// TIA Portal V18 export
// export: Created 2026-06-22T00:00:00Z, ExportSetting WithDefaults, DisplayName Totally Integrated Automation Portal, DisplayVersion V18
TagTable "Default tag table"
  CV3201_Nuoc_Bon1_M : Real  (PLC tag CV3201_Nuoc_Bon1_M, HMI_Connection_1, 1 s)   // Cảm biến/Van tuyến tính CV 32.01
  CV3206_Hoi_Bon2_M : Real  (PLC tag CV3206_Hoi_Bon2_M, HMI_Connection_1, 1 s)   // Cảm biến/Van tuyến tính CV 32.06
  CV3211_Nuoc_Bon3_M : Real  (PLC tag CV3211_Nuoc_Bon3_M, HMI_Connection_1, 1 s)   // Cảm biến/Van tuyến tính CV 32.11
  CV3216_Hoi_Bon4_M : Real  (PLC tag CV3216_Hoi_Bon4_M, HMI_Connection_1, 1 s)   // Cảm biến/Van tuyến tính CV 32.16
  CV3304_Nuoc_Lam_Mat_M : Real  (PLC tag CV3304_Nuoc_Lam_Mat_M, HMI_Connection_1, 1 s)   // Cảm biến/Van tuyến tính CV 33.04
  CV_Filler_Cap_Dich_M : Real  (PLC tag CV_Filler_Cap_Dich_M, HMI_Connection_1, 1 s)   // Cảm biến/Van tuyến tính CV Filler
  FQ3200_Bon1_Eff : Real  (PLC tag FQ3200_Bon1_Eff, HMI_Connection_1, 1 s)   // Cảm biến/Van tuyến tính FT 32.00
  FQ3205_Bon2_Eff : Real  (PLC tag FQ3205_Bon2_Eff, HMI_Connection_1, 1 s)   // Cảm biến/Van tuyến tính FT 32.05
  FQ3210_Bon3_Eff : Real  (PLC tag FQ3210_Bon3_Eff, HMI_Connection_1, 1 s)   // Cảm biến/Van tuyến tính FT 32.10
  FQ3215_Bon4_Eff : Real  (PLC tag FQ3215_Bon4_Eff, HMI_Connection_1, 1 s)   // Cảm biến/Van tuyến tính FT 32.15
  FT3309_Xa_Thanh_Pham_Eff : Real  (PLC tag FT3309_Xa_Thanh_Pham_Eff, HMI_Connection_1, 1 s)   // Cảm biến/Van tuyến tính FT 33.09
  HMI_Anim_Bon1_Frame : Int  (PLC tag HMI_Anim_Bon1_Frame, HMI_Connection_1, 1 s)   // Trạng thái hoạt hình HMI HMI_Anim_Bon1_Frame
  HMI_Anim_Bon1_MucDich : Int  (PLC tag HMI_Anim_Bon1_MucDich, HMI_Connection_1, 1 s)   // Trạng thái hoạt hình HMI HMI_Anim_Bon1_MucDich
  HMI_Anim_Bon2_Frame : Int  (PLC tag HMI_Anim_Bon2_Frame, HMI_Connection_1, 1 s)   // Trạng thái hoạt hình HMI HMI_Anim_Bon2_Frame
  HMI_Anim_Bon2_MucDich : Int  (PLC tag HMI_Anim_Bon2_MucDich, HMI_Connection_1, 1 s)   // Trạng thái hoạt hình HMI HMI_Anim_Bon2_MucDich
  HMI_Anim_Bon3_Frame : Int  (PLC tag HMI_Anim_Bon3_Frame, HMI_Connection_1, 1 s)   // Trạng thái hoạt hình HMI HMI_Anim_Bon3_Frame
  HMI_Anim_Bon3_MucDich : Int  (PLC tag HMI_Anim_Bon3_MucDich, HMI_Connection_1, 1 s)   // Trạng thái hoạt hình HMI HMI_Anim_Bon3_MucDich
  HMI_Anim_Bon4_Frame : Int  (PLC tag HMI_Anim_Bon4_Frame, HMI_Connection_1, 1 s)   // Trạng thái hoạt hình HMI HMI_Anim_Bon4_Frame
  HMI_Anim_Bon4_MucDich : Int  (PLC tag HMI_Anim_Bon4_MucDich, HMI_Connection_1, 1 s)   // Trạng thái hoạt hình HMI HMI_Anim_Bon4_MucDich
  HMI_Anim_BonChua1_MucDich : Int  (PLC tag HMI_Anim_BonChua1_MucDich, HMI_Connection_1, 1 s)   // Trạng thái hoạt hình HMI HMI_Anim_BonChua1_MucDich
  HMI_Anim_BonChua2_MucDich : Int  (PLC tag HMI_Anim_BonChua2_MucDich, HMI_Connection_1, 1 s)   // Trạng thái hoạt hình HMI HMI_Anim_BonChua2_MucDich
  LT3203_Bon1_Eff : Real  (PLC tag LT3203_Bon1_Eff, HMI_Connection_1, 1 s)   // Cảm biến/Van tuyến tính LT 32.03
  LT3209_Bon2_Eff : Real  (PLC tag LT3209_Bon2_Eff, HMI_Connection_1, 1 s)   // Cảm biến/Van tuyến tính LT 32.09
  LT3213_Bon3_Eff : Real  (PLC tag LT3213_Bon3_Eff, HMI_Connection_1, 1 s)   // Cảm biến/Van tuyến tính LT 32.13
  LT3218_Bon4_Eff : Real  (PLC tag LT3218_Bon4_Eff, HMI_Connection_1, 1 s)   // Cảm biến/Van tuyến tính LT 32.18
  LT3302_BonChua1_Eff : Real  (PLC tag LT3302_BonChua1_Eff, HMI_Connection_1, 1 s)   // Cảm biến/Van tuyến tính LT 33.02
  LT3307_BonChua2_Eff : Real  (PLC tag LT3307_BonChua2_Eff, HMI_Connection_1, 1 s)   // Cảm biến/Van tuyến tính LT 33.07
  PI3308_Truoc_Filter_Eff : Real  (PLC tag PI3308_Truoc_Filter_Eff, HMI_Connection_1, 1 s)   // Cảm biến/Van tuyến tính PI 33.08
  Pump3264_Chuyen_Nhanh1_M : Bool  (PLC tag Pump3264_Chuyen_Nhanh1_M, HMI_Connection_1, 1 s)   // Trạng thái hoạt động Pump 32.64
  Pump3265_Chuyen_Nhanh2_M : Bool  (PLC tag Pump3265_Chuyen_Nhanh2_M, HMI_Connection_1, 1 s)   // Trạng thái hoạt động Pump 32.69
  Pump3361_LuanChuyen_BonChua1_M : Bool  (PLC tag Pump3361_LuanChuyen_BonChua1_M, HMI_Connection_1, 1 s)   // Trạng thái hoạt động Pump 33.61
  Pump3362_Xa_BonChua1_M : Bool  (PLC tag Pump3362_Xa_BonChua1_M, HMI_Connection_1, 1 s)   // Trạng thái hoạt động Pump 33.62
  Pump3364_Filter_M : Bool  (PLC tag Pump3364_Filter_M, HMI_Connection_1, 1 s)   // Trạng thái hoạt động Pump 33.64
  Pump3365_Filter_M : Bool  (PLC tag Pump3365_Filter_M, HMI_Connection_1, 1 s)   // Trạng thái hoạt động Pump 33.65
  TT3204_Bon1_Eff : Real  (PLC tag TT3204_Bon1_Eff, HMI_Connection_1, 1 s)   // Cảm biến/Van tuyến tính TT 32.04
  TT3208_Bon2_Eff : Real  (PLC tag TT3208_Bon2_Eff, HMI_Connection_1, 1 s)   // Cảm biến/Van tuyến tính TT 32.08
  TT3214_Bon3_Eff : Real  (PLC tag TT3214_Bon3_Eff, HMI_Connection_1, 1 s)   // Cảm biến/Van tuyến tính TT 32.14
  TT3219_Bon4_Eff : Real  (PLC tag TT3219_Bon4_Eff, HMI_Connection_1, 1 s)   // Cảm biến/Van tuyến tính TT 32.19
  TT3301_BonChua1_Eff : Real  (PLC tag TT3301_BonChua1_Eff, HMI_Connection_1, 1 s)   // Cảm biến/Van tuyến tính TT 33.01
  TT3303_TraoDoiNhiet_Eff : Real  (PLC tag TT3303_TraoDoiNhiet_Eff, HMI_Connection_1, 1 s)   // Cảm biến/Van tuyến tính TT 33.03
  TT3306_BonChua2_Eff : Real  (PLC tag TT3306_BonChua2_Eff, HMI_Connection_1, 1 s)   // Cảm biến/Van tuyến tính TT 33.06
  V3230_Nuoc_Bon1_M : Bool  (PLC tag V3230_Nuoc_Bon1_M, HMI_Connection_1, 1 s)   // Trạng thái hoạt động V32.30
  V3232_Xa_Bon1_M : Bool  (PLC tag V3232_Xa_Bon1_M, HMI_Connection_1, 1 s)   // Trạng thái hoạt động V32.32
  V3233_Xa_Bon1_M : Bool  (PLC tag V3233_Xa_Bon1_M, HMI_Connection_1, 1 s)   // Trạng thái hoạt động V32.33
  V3234_Xa_Bon1_M : Bool  (PLC tag V3234_Xa_Bon1_M, HMI_Connection_1, 1 s)   // Trạng thái hoạt động V32.34
  V3235_Nuoc_Bon2_M : Bool  (PLC tag V3235_Nuoc_Bon2_M, HMI_Connection_1, 1 s)   // Trạng thái hoạt động V32.35
  V3237_Xa_Bon2_M : Bool  (PLC tag V3237_Xa_Bon2_M, HMI_Connection_1, 1 s)   // Trạng thái hoạt động V32.37
  V3238_Xa_Bon2_M : Bool  (PLC tag V3238_Xa_Bon2_M, HMI_Connection_1, 1 s)   // Trạng thái hoạt động V32.38
  V3239_Xa_Bon2_M : Bool  (PLC tag V3239_Xa_Bon2_M, HMI_Connection_1, 1 s)   // Trạng thái hoạt động V32.39
  V3240_Nuoc_Bon3_M : Bool  (PLC tag V3240_Nuoc_Bon3_M, HMI_Connection_1, 1 s)   // Trạng thái hoạt động V32.40
  V3242_Xa_Bon3_M : Bool  (PLC tag V3242_Xa_Bon3_M, HMI_Connection_1, 1 s)   // Trạng thái hoạt động V32.42
  V3243_Xa_Bon3_M : Bool  (PLC tag V3243_Xa_Bon3_M, HMI_Connection_1, 1 s)   // Trạng thái hoạt động V32.43
  V3244_Xa_Bon3_M : Bool  (PLC tag V3244_Xa_Bon3_M, HMI_Connection_1, 1 s)   // Trạng thái hoạt động V32.44
  V3245_Nuoc_Bon4_M : Bool  (PLC tag V3245_Nuoc_Bon4_M, HMI_Connection_1, 1 s)   // Trạng thái hoạt động V32.45
  V3247_Xa_Bon4_M : Bool  (PLC tag V3247_Xa_Bon4_M, HMI_Connection_1, 1 s)   // Trạng thái hoạt động V32.47
  V3248_Xa_Bon4_M : Bool  (PLC tag V3248_Xa_Bon4_M, HMI_Connection_1, 1 s)   // Trạng thái hoạt động V32.48
  V3249_Xa_Bon4_M : Bool  (PLC tag V3249_Xa_Bon4_M, HMI_Connection_1, 1 s)   // Trạng thái hoạt động V32.49
  V3331_Xa_BonChua1_M : Bool  (PLC tag V3331_Xa_BonChua1_M, HMI_Connection_1, 1 s)   // Trạng thái hoạt động V33.31
  V3332_Xa_BonChua1_M : Bool  (PLC tag V3332_Xa_BonChua1_M, HMI_Connection_1, 1 s)   // Trạng thái hoạt động V33.32
  V3333_DieuHuong_BonChua1_M : Bool  (PLC tag V3333_DieuHuong_BonChua1_M, HMI_Connection_1, 1 s)   // Trạng thái hoạt động V33.33
  V3334_DieuHuong_BonChua1_M : Bool  (PLC tag V3334_DieuHuong_BonChua1_M, HMI_Connection_1, 1 s)   // Trạng thái hoạt động V33.34
  V3335_DieuHuong_BonChua1_M : Bool  (PLC tag V3335_DieuHuong_BonChua1_M, HMI_Connection_1, 1 s)   // Trạng thái hoạt động V33.35
  V3338_Xa_BonChua2_M : Bool  (PLC tag V3338_Xa_BonChua2_M, HMI_Connection_1, 1 s)   // Trạng thái hoạt động V33.38
  V3339_Xa_BonChua2_M : Bool  (PLC tag V3339_Xa_BonChua2_M, HMI_Connection_1, 1 s)   // Trạng thái hoạt động V33.39
  V3340_Duong_Filter_M : Bool  (PLC tag V3340_Duong_Filter_M, HMI_Connection_1, 1 s)   // Trạng thái hoạt động V33.40
  V3341_Duong_Filter_M : Bool  (PLC tag V3341_Duong_Filter_M, HMI_Connection_1, 1 s)   // Trạng thái hoạt động V33.41
